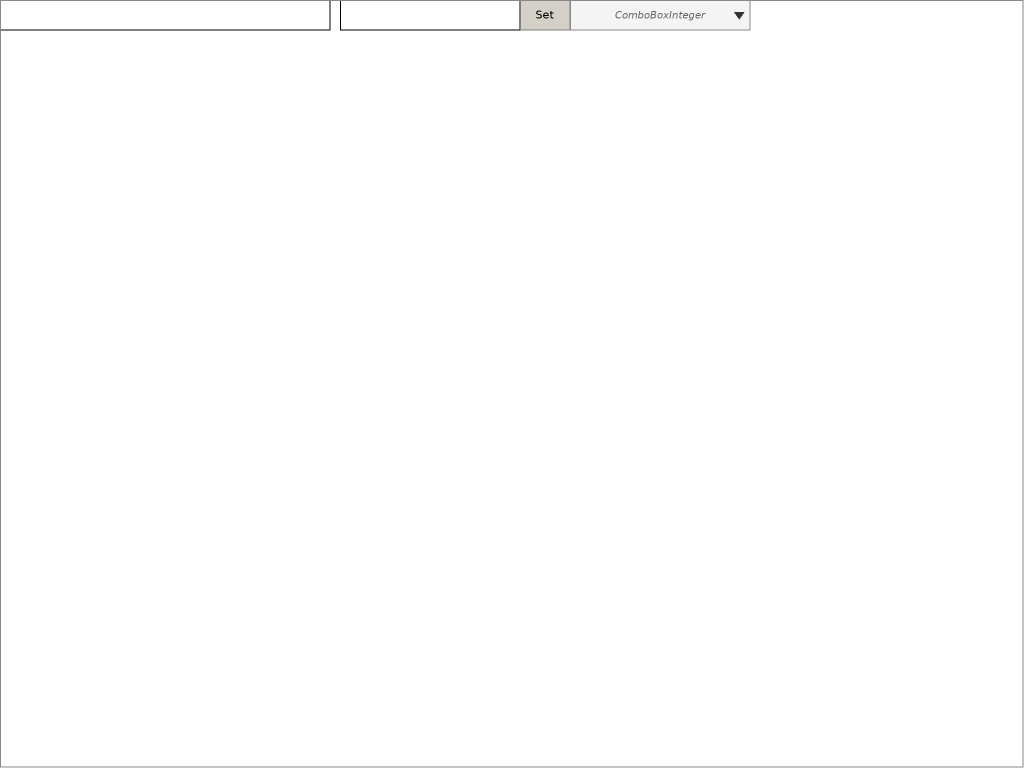
VISUALIZATION Param_ENUM_TermType  // 1024x768
    Rectangle (340,0 180x30), text list: 'TL_TerminalType', text index: stMParam_Visu.nEnumAktValue[nIdx]
    Rectangle (0,0 330x30), text list: 'TL_Params_Enum', text index: nIdx
    Rectangle (520,0 50x30), "Set"
        OnMouseClick: execute { stMParam_Visu.bEnumSetValue[nIdx]:=TRUE; }
    ComboBoxInteger (570,0 180x30), variable: stMParam_Visu.nEnumNewValue[nIdx], text list: 'TL_TerminalType'
END_VISUALIZATION

(* stored: Version 1.1.0.1
   Visu Param_ENUM_TermType: Id {9ee2d918-8691-495a-92a6-97cf7d7dd3b2} *)
